PROGRAM LEDs
VAR	
	Red		AT%Q*	:	INT;
	Green	AT%Q*	:	INT;
	Blue	AT%Q*	:	INT;
	White	AT%Q*	:	INT;
	
	countdown	:	Countdown;
END_VAR

countdown(RedOut => Red,GreenOut => Green, BlueOut => Blue,WhiteOut => White);

END_PROGRAM

(* stored: Version 1.1.0.1, ProductVersion 3.1.4024.12
   POU LEDs: Id {080668ae-5330-4f9e-94a4-ce20fb139d33}, SpecialFunc None *)
